{attribute 'qualified_only'}
{attribute 'strict'}
TYPE E_SeqState :
(
	STANDBY, 
	WRITE_REQ, 
	WRITE_WAIT, 
	COUNTDOWN, 
	EXECUTE
);
END_TYPE

(* stored: Version 1.1.0.1, ProductVersion 3.1.4024.15
   DUT E_SeqState: Id {4c68ae9f-f959-4048-a4d9-2bb7cb06e6e5} *)
